TYPE FiberSwitchConfigs :
STRUCT
	EOLFiberSwitchConfig : EOLFiberSwitchConfig;
END_STRUCT
END_TYPE

(* stored: Version 1.1.0.1, ProductVersion 3.1.4024.3
   DUT FiberSwitchConfigs: Id {a91366a1-630f-4a2d-a61c-f4efee732494} *)
